TEXTLIST CRAH_Status
  0 = 'Hand'
  1 = 'Off'
  2 = 'Auto'
   = ''
END_TEXTLIST

(* stored: Version 1.1.0.1, ProductVersion 3.1.4024.12
   TextList CRAH_Status: Id {8c48fc8a-b556-4397-a3f0-48059c892dde} *)
